TYPE VTD_Inputs_DUT :
STRUCT
	Upper_Overtravel:  BOOL;
	Upper_limit:  BOOL;
	Ultimate_SlowDown:  Bool;
	Ultimate_Creep:  Bool;
	Lower_Limit:  Bool;
	Lower_Overtravel:  Bool;
	Level_Detect1:  Bool;
	Level_Detect2:  BOOL;
	DP1_Extended:  BOOL;
	DP2_Extended:  BOOL;
	DP1_Retracted:  BOOL;
	DP2_Retracted:  Bool;
	Chain_Slack_1:  Bool;
	Chain_Slack_2:  Bool;
	Chain_Slack_3:  Bool;
	Chain_Slack_4:  Bool;
	PushToEnter:  Bool;
	PushToExit:  Bool;
	Barcode_1:  STRING;
	Barcode_2:  STRING;
	LE_Status:  UInt;
	LE_Position:  DInt;
	LE_Speed:  Int;
	LE_Warnings:  Int;
	LE_Quality_Decoded_Codes:  Byte;
	LE_Quality_Value:  Byte;
	AE_Status_1:  UInt;
	AE_Status_2:  UInt;
	AE_Position_1:  DInt;
	AE_Position_2:  DInt;
	AE_Speed:  Int;
	VFD_Status:  Word;
	VFD_Speed_Actual:  Word;
	VFD_ActualCurrent:  Int;
	VFD_ActualTorque:  INT;
END_STRUCT
END_TYPE

(* stored: Version 1.1.0.1
   DUT VTD_Inputs_DUT: Id {5b8d14b2-9176-4a98-95bc-d13a5d1e0512} *)
